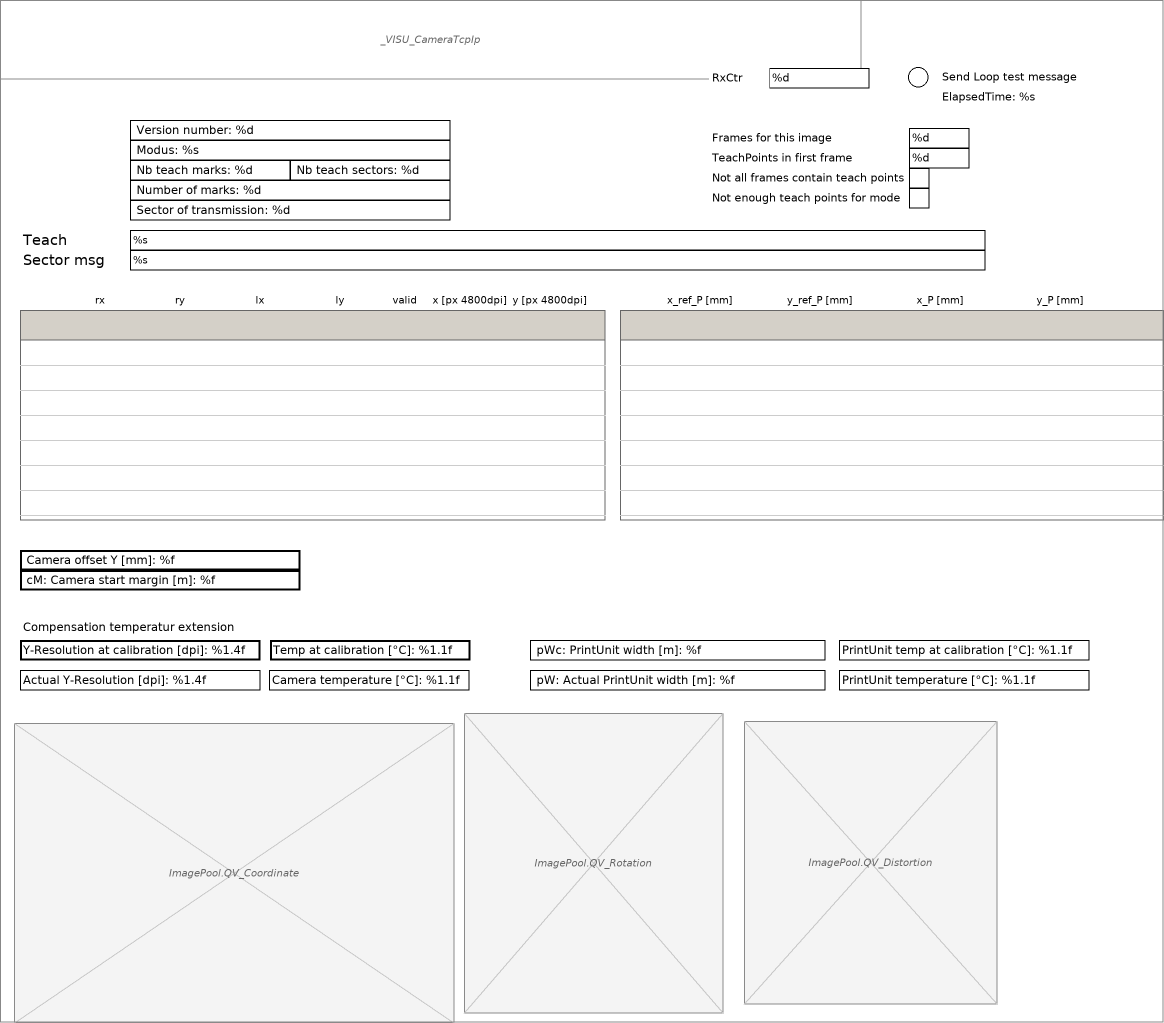
VISUALIZATION _VISU_LineCamera  // 1164x1023
VAR_INPUT
	m_Inst : FB_LineCamera;
END_VAR
    Rectangle (20,230 100x20), "Teach"
    Rectangle (130,230 855x20), "%s", text variable: m_Inst.sTeach
    Rectangle (130,120 320x20), "Version number: %d", text variable: m_Inst.nNbVersion
    Rectangle (130,160 160x20), "Nb teach marks: %d", text variable: m_Inst.nNbMarksTeach
    Table (20,310 585x210), data array: m_Inst.sCameraPoints
        p1128707560: GVL_Camera.cMaxNbMarks
        p2501879983: m_Inst.stCameraResult[INDEX].y_ref_Print
        p7306298: m_Inst.stCameraResult[INDEX].x_teach_Print
        p1933151965: m_Inst.stCameraResult[INDEX].y_teach_Print
        p3863566920: m_Inst.stCameraResult[INDEX].x_Print
        p2192122294: m_Inst.stCameraResult[INDEX].y_Print
        p3854506369: m_Inst.sCameraPoints[INDEX].id
        p1892666644: m_Inst.sCameraPoints[INDEX].x_ref
        p338671338: m_Inst.sCameraPoints[INDEX].y_ref
        p2170511999: m_Inst.sCameraPoints[INDEX].lx
        p3723444502: m_Inst.sCameraPoints[INDEX].ly
        p1218418051: m_Inst.sCameraPoints[INDEX].valid
    Rectangle (60,290 80x20), "rx"
    Rectangle (140,290 80x20), "ry"
    Rectangle (220,290 80x20), "lx"
    Rectangle (300,290 80x20), "ly"
    Rectangle (430,290 80x20), "x [px 4800dpi]"
    Rectangle (510,290 80x20), "y [px 4800dpi]"
    Rectangle (380,290 50x20), "valid"
    Rectangle (130,200 320x20), "Sector of transmission: %d", text variable: m_Inst.nSector
    Rectangle (530,640 295x20), "pWc: PrintUnit width [m]: %f", text variable: m_Inst._fPrintUnitWidthTC
    Image (14,723 440x300), image: ImagePool.QV_Coordinate
    Image (464,713 259x300), image: ImagePool.QV_Rotation
    Image (744,721 253x283), image: ImagePool.QV_Distortion
    Rectangle (20,250 100x20), "Sector msg"
    Rectangle (130,250 855x20), "%s", text variable: m_Inst.sMemLastMessage
    Rectangle (660,290 80x20), "x_ref_P [mm]"
    Rectangle (780,290 80x20), "y_ref_P [mm]"
    Rectangle (900,290 80x20), "x_P [mm]"
    Rectangle (1020,290 80x20), "y_P [mm]"
    Table (620,310 544x210), data array: m_Inst.sTeachPoints
        p1128707560: GVL_Camera.cMaxNbMarks
        p746581629: m_Inst.stCameraResult[INDEX].y
        p3104783080: m_Inst.stCameraResult[INDEX].x_ref_Print
        p2501879983: m_Inst.stCameraResult[INDEX].y_ref_Print
        p7306298: m_Inst.stCameraResult[INDEX].x_teach_Print
        p1933151965: m_Inst.stCameraResult[INDEX].y_teach_Print
        p3863566920: m_Inst.stCameraResult[INDEX].x_Print
        p2192122294: m_Inst.stCameraResult[INDEX].y_Print
        p3854506369: m_Inst.sTeachPoints[INDEX].x_ref_Print
        p1892666644: m_Inst.sTeachPoints[INDEX].y_ref_Print
        p338671338: m_Inst.sTeachPoints[INDEX].x_teach_Print
        p2170511999: m_Inst.sTeachPoints[INDEX].y_teach_Print
        p3723444502: m_Inst.sTeachPoints[INDEX].x_Print
        p1218418051: m_Inst.sTeachPoints[INDEX].y_Print
    Rectangle (20,640 240x20), "Y-Resolution at calibration [dpi]: %1.4f", text variable: m_Inst.fCameraResolution
        OnMouseDown: write the text variable via Edit
    Rectangle (20,670 240x20), "Actual Y-Resolution [dpi]: %1.4f", text variable: m_Inst.fCameraRealResolution
    Rectangle (269,670 200x20), "Camera temperature [°C]: %1.1f", text variable: m_Inst.fCameraTemp
    Rectangle (270,640 200x20), "Temp at calibration [°C]: %1.1f", text variable: m_Inst.fCameraCalTemp
        OnMouseDown: write the text variable via Edit
    Rectangle (839,640 250x20), "PrintUnit temp at calibration [°C]: %1.1f", text variable: m_Inst._fPrintUnitCalTemp
    Rectangle (839,670 250x20), "PrintUnit temperature [°C]: %1.1f", text variable: m_Inst.fPrintUnitTemp
    Rectangle (20,617 245x20), "Compensation temperatur extension"
    Rectangle (530,670 295x20), "pW: Actual PrintUnit width [m]: %f", text variable: m_Inst.fPrintUnitWidthTAct
    Rectangle (130,180 320x20), "Number of marks: %d", text variable: m_Inst.nNbMarks
    Rectangle (20,550 280x20), "Camera offset Y [mm]: %f", text variable: m_Inst.fCameraAdjustmentY
        OnMouseDown: write the text variable via Edit
    Rectangle (20,570 280x20), "cM: Camera start margin [m]: %f", text variable: m_Inst.fCameraStartMargin
        OnMouseDown: write the text variable via Edit
    Rectangle (130,140 320x20), "Modus: %s", text variable: m_Inst.sModus
    Frame (0,0 861x79)
        shows _VISU_CameraTcpIp(m_Inst := m_Inst)
    Rectangle (290,160 160x20), "Nb teach sectors: %d", text variable: m_Inst.nNbSectorTeach
    Ellipse (908,67 20x20)
        tap m_Inst._bTestTx
    Rectangle (769,68 100x20), "%d", text variable: m_Inst.nRxMsg
    Rectangle (709,68 60x20), "RxCtr"
    Rectangle (939,67 161x20), "Send Loop test message"
    Rectangle (939,87 161x20), "ElapsedTime: %s", text variable: m_Inst._sTimeElapsed
    Rectangle (709,128 200x20), "Frames for this image"
    Rectangle (909,128 60x20), "%d", text variable: m_Inst.nNumFrames
    Rectangle (709,148 200x20), "TeachPoints in first frame"
    Rectangle (909,148 60x20), "%d", text variable: m_Inst.nNumPointsPerSectorT[1]
    Rectangle (709,168 200x20), "Not all frames contain teach points"
    RoundedRectangle (909,168 20x20), colour toggle: m_Inst.bNotAllFramesContainTeachPoints
    Rectangle (709,188 200x20), "Not enough teach points for mode"
    RoundedRectangle (909,188 20x20), colour toggle: m_Inst.bNotEnoughTeachPoints
END_VISUALIZATION

(* stored: Version 1.1.0.1, ProductVersion 3.1.4024.3
   Visu _VISU_LineCamera: Id {e1331a9c-9add-4ea7-b07b-32215c09bb03} *)
